{attribute 'linkalways'} 
{attribute 'no_explicit_call' := 'This FB is a CLASS and must be accessed using methods or properties'}
{attribute 'enable_dynamic_creation'}
FUNCTION_BLOCK _TIME_OF_DAY EXTENDS DatatypeBase
VAR
	localData : TIME_OF_DAY;
	activeData : REFERENCE TO TIME_OF_DAY REF= localData;
END_VAR

PROPERTY PUBLIC Address : PVOID
GET
Address := ADR(activeData);
END_GET
END_PROPERTY

METHOD PUBLIC ClearReference
VAR_INPUT
END_VAR
activeData REF= localData;
END_METHOD

METHOD PUBLIC Clone : I_Datatype
VAR
    pClone : POINTER TO _TIME_OF_DAY;
END_VAR
pClone := __NEW(_TIME_OF_DAY(InitialValue := Value));
Clone := pClone^;
END_METHOD

METHOD FB_init : BOOL
VAR_INPUT
	bInitRetains : BOOL; // if TRUE, the retain variables are initialized (warm start / cold start)
	bInCopyCode : BOOL;  // if TRUE, the instance afterwards gets moved WORDo the copy code (online change)
	InitialValue : TIME_OF_DAY;
END_VAR
localData := InitialValue;
END_METHOD

METHOD PUBLIC MakeReferenceTo
VAR_INPUT
	ReferenceTarget : REFERENCE TO TIME_OF_DAY;
END_VAR
activeData REF= ReferenceTarget;
END_METHOD

METHOD PUBLIC SerializeWith
VAR_INPUT
	Serializer : I_Serializer;
END_VAR
Serializer.AddTod(activeData);
END_METHOD

PROPERTY PUBLIC Size : UDINT
GET
Size := SIZEOF(activeData);
END_GET
END_PROPERTY

METHOD TryDeserializeFrom : BOOL
VAR_INPUT
	Deserializer : I_Deserializer;
	Feedback : I_DeserializerFeedback;
END_VAR
TryDeserializeFrom := Deserializer.TryGetTod(activeData, Feedback);
END_METHOD

METHOD TryMakeReferenceTo : BOOL
VAR_INPUT
	Target : I_Datatype;
END_VAR
VAR
	pTargetData : POINTER TO TIME_OF_DAY;
END_VAR
IF NOT (Target.TypeName = TypeName) THEN
	RETURN;
END_IF

pTargetData := Target.Address;
activeData REF= pTargetData^;
TryMakeReferenceTo := TRUE;
END_METHOD

PROPERTY PUBLIC TypeName : T_MAXSTRING
GET
TypeName := 'TIME_OF_DAY';
END_GET
END_PROPERTY

PROPERTY PUBLIC Value : TIME_OF_DAY
GET
Value := activeData;
END_GET
SET
activeData := Value;
END_SET
END_PROPERTY

END_FUNCTION_BLOCK

(* stored: Version 1.1.0.1, ProductVersion 3.1.4024.12
   POU _TIME_OF_DAY: Id {e38e9ffe-eab5-401f-8d8e-cef1ac28ee89}, SpecialFunc None
   Folder Constructor: Id {56f24a88-7864-453a-9028-aaf46bcf2fc4}
   Property Address: Id {7d9d061c-5328-428f-9bc1-3c06a45be2be}
   Get Get: Id {a935aad8-2c2c-4446-8e67-6208185c353a}
   Method ClearReference: Id {0dae4100-1f0f-4f49-b5f9-368bd7f40aef}
   Method Clone: Id {620e6105-7f31-4609-9c08-f7a7dd5c86ce}
   Method FB_init: Id {b739d7d2-98be-4ec7-934e-63da4c4cb534}
   Method MakeReferenceTo: Id {24ba2d59-aedf-4da3-b88d-e796575bbb80}
   Method SerializeWith: Id {9ac5d77e-210e-46d5-8d10-4d0d0a0e28a1}
   Property Size: Id {d498b416-736d-4d2d-a706-97e8f7ee1e47}
   Get Get: Id {162c049e-768e-451e-ab65-4e4530f42031}
   Method TryDeserializeFrom: Id {40c6d612-a4d5-4177-a108-d8d5561dc5e3}
   Method TryMakeReferenceTo: Id {8ffde550-2da4-4810-9db5-b0fb562c29df}
   Property TypeName: Id {350e728a-0d27-4e5b-a300-5cd44f55dfb3}
   Get Get: Id {1dd882e1-2db0-4345-a274-1f1ccf266e83}
   Property Value: Id {8a5f6f50-27b5-4f48-aedb-9075d7668289}
   Get Get: Id {86833ed5-82ad-4956-9d8e-51282191da28}
   Set Set: Id {2ca3a9e6-d409-4e66-9d85-1d34812cd70d} *)
